// TIA Portal V17 export
// export: Created 2025-06-26T06:49:27.5294256Z, ExportSetting WithDefaults, DisplayName Totally Integrated Automation Portal, DisplayVersion V17 Update 8, DisplayName TIA Portal Openness, DisplayVersion V17 Update 8, DisplayName TIA Portal Version Control Interface, DisplayVersion V17, DisplayName STEP 7 Professional, DisplayVersion V17 Update 8, DisplayName STEP 7 Safety, DisplayVersion V17 Update 6, DisplayName WinCC Advanced, DisplayVersion V17 Update 8
TYPE "stProfile"
// stored: IsFailsafeCompliant false
   STRUCT
      lfMemory : LReal;   // Internal state
      lfElapsed : LReal;   // Profile value
   END_STRUCT;
END_TYPE
